(* CODESYS project FU_sDeleteRight.xml

Project tree, tasks and I/O mapping:
  function FU_sDeleteRight [ST]
*)

// FU_sDeleteRight
//This functions deletes a part of a string values are counted from the right instead of the left
// +-----------+----------+----------+-----------------------------------------------------------------------------------------------------------------------+
// |**Version**|**Author**| **Date** |**Changes**                                                                                                            |
// +-----------+----------+----------+-----------------------------------------------------------------------------------------------------------------------+
// | 1         | NSN      | 22-02-19 | Creation                                                                                                              |
// +-----------+----------+----------+-----------------------------------------------------------------------------------------------------------------------+
FUNCTION FU_sDeleteRight : STRING(255)
VAR_INPUT
	sStr		:STRING(255);		//Input String
	wLen		:WORD;				//Amount to delete
	wPos		:WORD;				//Position to delete from
END_VAR

FU_sDeleteRightBIBO(sOut:= FU_sDeleteRight, sStr:= sStr, wLen:= wLen,wPos:= wPos, wOutSize:= 255);

END_FUNCTION
